INTERFACE I_MonoSymbol EXTENDS I_Symbol

PROPERTY PUBLIC BackgroundColor : Pixel
GET
END_GET
SET
END_SET
END_PROPERTY

PROPERTY PUBLIC ForgroundColor : Pixel
GET
END_GET
SET
END_SET
END_PROPERTY

METHOD PUBLIC InvertColor
VAR_INPUT
END_VAR
END_METHOD

END_INTERFACE

(* stored: Version 1.1.0.1, ProductVersion 3.1.4024.15
   Itf I_MonoSymbol: Id {1813fd47-3e7a-4b74-95bc-f71ea72690ff}
   Property BackgroundColor: Id {ef9693ec-801c-48f6-9658-b92558797f91}
   Get Get: Id {c6a57c36-f26f-4690-ba93-c8eaf9cc2bd8}
   Set Set: Id {d5d2c8cc-22d6-41a7-8b63-e12c1016fc09}
   Property ForgroundColor: Id {d202bc22-246d-4951-b274-45b865d0230c}
   Get Get: Id {a714be56-9f09-425a-8340-b289ff68b733}
   Set Set: Id {e25eea17-fe7e-4ca9-9230-b1fa516f58f0}
   Method InvertColor: Id {ca967492-af25-4a23-9511-2e7f4f31b36b} *)
